// TwinCAT 3 PLC project _01_Observer
// ProgramVersion: 3.1.4023.0
// libraries:
//   Tc2_Standard, * (Beckhoff Automation GmbH)
//   Tc2_System, * (Beckhoff Automation GmbH)
//   Tc3_Module, * (Beckhoff Automation GmbH)
// project tree:
//   / MAIN.TcPOU, PlcTask.TcTTO
//   Observer Pattern/Pattern Base/ I_Observable.TcIO, I_Observer.TcIO, Observable.TcPOU
//   Observer Pattern/ P_ObserverPattern.TcPOU
//   Observer Pattern/Samples/ EventPublisherWithInheritance.TcPOU, EventPublisherWithComposition.TcPOU, FB_EventSubscriber.TcPOU, FB_EventSubscriber2.TcPOU, I_EventPublisher.TcIO
// (motion and I/O tree: see PLC project 13_decorator)
// real-time tasks:
//   TASK PlcTask: cycle T#10ms, priority 20, ADS port 350
// variable links:

CONFIGURATION _01_Observer
    RESOURCE PLC ON TwinCAT3
        TASK PlcTask(INTERVAL := T#10ms, PRIORITY := 20);
        PROGRAM MAIN WITH PlcTask : MAIN;
    END_RESOURCE
END_CONFIGURATION

// ---- Observer Pattern/Pattern Base/I_Observable.TcIO
INTERFACE I_Observable

METHOD Attach : bool
VAR_INPUT
	observer			: I_Observer;
END_VAR
END_METHOD

METHOD Detach : BOOL
VAR_INPUT
	observer			: I_Observer;
END_VAR
END_METHOD

END_INTERFACE

// ---- Observer Pattern/Pattern Base/I_Observer.TcIO
INTERFACE I_Observer

METHOD Update : BOOL
VAR_INPUT
END_VAR
END_METHOD

END_INTERFACE

// ---- Observer Pattern/Samples/I_EventPublisher.TcIO
INTERFACE I_EventPublisher EXTENDS I_Observable

PROPERTY Event : int
GET
END_GET
END_PROPERTY

END_INTERFACE

// ---- MAIN.TcPOU
PROGRAM MAIN
VAR
END_VAR

(* 
	GOF 		Define a one-to-many dependency between objects so that when one object changes state, 
				all its dependents are notified and updated automatically   
*)
P_ObserverPattern();

END_PROGRAM

// ---- Observer Pattern/P_ObserverPattern.TcPOU
PROGRAM P_ObserverPattern
VAR
	eventPublisher					: EventPublisherWithInheritance;
	eventPublisher2					: EventPublisherWithComposition;	
	
	eventSubscriber					: FB_EventSubscriber(eventPublisher);	
	eventSubscriber2				: FB_EventSubscriber2(eventPublisher2);	
	
	triggerEvent					: BOOL;
END_VAR

// Property changeEvent was only to be able to change the event from outside for the unit test
// Change according the use case of the observer
IF triggerEvent	THEN
	eventPublisher.changeEvent := eventPublisher.event + 1;
	eventPublisher2.changeEvent := eventPublisher2.event + 1;
	triggerEvent := FALSE;
END_IF
eventPublisher.CyclicCall();
eventPublisher2.CyclicCall();
eventSubscriber.CyclicCall();
eventSubscriber2.CyclicCall();

END_PROGRAM

// ---- Observer Pattern/Samples/EventPublisherWithInheritance.TcPOU
{attribute 'no_explicit_call' := 'FB_EventPublisher is a CLASS and must be accessed using methods or properties'}
FUNCTION_BLOCK EventPublisherWithInheritance EXTENDS Observable IMPLEMENTS I_EventPublisher
VAR
	_event							: INT;
	eventPrev						: INT;
END_VAR


// The body of a class must not be used for code.  
// Cyclic code should be called from a method if needed.

PROPERTY PUBLIC ChangeEvent : int
SET
// IMPLEMENTED ONLY FOR TESTING PURPOSES
VAR
END_VAR
_event := changeEvent;
END_SET
END_PROPERTY

METHOD CyclicCall
IF eventPrev <> _event 			THEN
	notify();
	eventPrev := _event;
END_IF
END_METHOD

// IMPLEMENTED ONLY FOR TESTING PURPOSES
PROPERTY Event : int
GET
event := _event;
END_GET
END_PROPERTY

END_FUNCTION_BLOCK

// ---- Observer Pattern/Pattern Base/Observable.TcPOU
{attribute 'no_explicit_call' := 'Observable is a CLASS and must be accessed using methods or properties'}
FUNCTION_BLOCK Observable IMPLEMENTS I_Observable
VAR
	verbose							: BOOL := TRUE;
	observers						: ARRAY[1..MAXOBSERVERS] OF I_Observer;
END_VAR
VAR CONSTANT
	MAXOBSERVERS					: INT := 5;		
END_VAR


// The body of a class must not be used for code.  
// Cyclic code should be called from a method if needed.

METHOD attach : BOOL
VAR_INPUT
	observer			: I_Observer;
END_VAR
VAR
	i					: INT;
END_VAR
(* default *)
attach := FALSE;

(* loop if the subscriber is already registered *)
FOR i := 1 TO MAXOBSERVERS DO
	IF observers[i] = observer 	THEN
		observer.update();
		attach := TRUE;
		RETURN;
	END_IF
END_FOR

(* loop for first free position if not yet attached *)
FOR i := 1 TO MAXOBSERVERS DO
	IF observers[i] = 0 	THEN
		observers[i] := observer;
		message('Observer registered');
		observer.update();
		attach := TRUE;
		EXIT;
	END_IF
END_FOR
END_METHOD

METHOD detach : BOOL
VAR_INPUT
	observer			: I_Observer;
END_VAR
VAR
	i					: INT;
END_VAR
(* default *)
detach := FALSE;

(* loop if the subscriber is already registered *)
FOR i := 1 TO MAXOBSERVERS DO
	IF observers[i] = observer 	THEN
		observers[i] := 0;
		message('Observer deregistered');
		detach := TRUE;
		RETURN;
	END_IF
END_FOR
END_METHOD

METHOD PRIVATE message : BOOL
VAR_INPUT
	strArg						: STRING;
END_VAR
// Log message
IF verbose  THEN
	ADSLOGSTR(
		msgCtrlMask := ADSLOG_MSGTYPE_HINT OR ADSLOG_MSGTYPE_LOG, // ADSLOG_MSGTYPE_ERROR OR ADSLOG_MSGTYPE_LOG, 
		msgFmtStr 	:= '%s',
		strArg 		:= strArg
		);
END_IF
END_METHOD

PROPERTY noOfAttachedObservers : int
GET
VAR
	i							: INT;
END_VAR
// In stead of using an internal counter that could fail
// run through the array of attached observers
(* loop for first free position if not yet attached *)
NoOfAttachedObservers := 0;
FOR i := 1 TO MAXOBSERVERS DO
	IF observers[i] <> 0 	THEN
		NoOfAttachedObservers := NoOfAttachedObservers + 1;
	END_IF
END_FOR
END_GET
END_PROPERTY

METHOD notify : BOOL
VAR
	i			: INT;
END_VAR
(* default *)
notify := FALSE;

(* loop if the subscriber is already registered *)
FOR i := 1 TO MAXOBSERVERS DO
	IF observers[i] <> 0 	THEN
		observers[i].update();
	END_IF
END_FOR
END_METHOD

END_FUNCTION_BLOCK

// ---- Observer Pattern/Samples/EventPublisherWithComposition.TcPOU
{attribute 'no_explicit_call' := 'FB_EventPublisher is a CLASS and must be accessed using methods or properties'}
FUNCTION_BLOCK EventPublisherWithComposition IMPLEMENTS I_EventPublisher
VAR
	_event							: INT;
	eventPrev						: INT;
	
	observable						: Observable;
END_VAR


// The body of a class must not be used for code.  
// Cyclic code should be called from a method if needed.

METHOD Attach : BOOL
VAR_INPUT
	observer	: I_Observer;
END_VAR
Attach := observable.Attach(observer);
END_METHOD

PROPERTY PUBLIC ChangeEvent : int
SET
// IMPLEMENTED ONLY FOR TESTING PURPOSES
VAR
END_VAR
_event := changeEvent;
END_SET
END_PROPERTY

METHOD CyclicCall
IF eventPrev <> _event 			THEN
	observable.Notify();
	eventPrev := _event;
END_IF
END_METHOD

METHOD Detach : BOOL
VAR_INPUT
	observer	: I_Observer;
END_VAR
Detach := observable.Detach(observer);
END_METHOD

// IMPLEMENTED ONLY FOR TESTING PURPOSES
PROPERTY Event : int
GET
event := _event;
END_GET
END_PROPERTY

END_FUNCTION_BLOCK

// ---- Observer Pattern/Samples/FB_EventSubscriber.TcPOU
{attribute 'no_explicit_call' := 'FB_EventSubscriber is a CLASS and must be accessed using methods or properties'}
FUNCTION_BLOCK FB_EventSubscriber IMPLEMENTS I_Observer
VAR	
	_eventPublisher					: I_EventPublisher;
	_event							: INT;
	
	verbose							: BOOL := TRUE;

	// Register after online change 
	registeredAtPublisher			: BOOL;	
END_VAR


// The body of a class must not be used for code.  
// Cyclic code should be called from a method if needed.

METHOD ChangePublisher
VAR_INPUT
	eventPublisher					: I_EventPublisher;
END_VAR
_eventPublisher := eventPublisher;
END_METHOD

METHOD cyclicCall
// Did we already register in the publisher?
IF NOT registeredAtPublisher	THEN
	registeredAtPublisher := _eventPublisher.attach(THIS^);
END_IF
END_METHOD

// IMPLEMENTED ONLY FOR TESTING PURPOSES
PROPERTY Event : int
GET
event := _event;
END_GET
END_PROPERTY

METHOD FB_init : BOOL
VAR_INPUT
	bInitRetains	 				: BOOL; // if TRUE, the retain variables are initialized (warm start / cold start)
	bInCopyCode 					: BOOL;  // if TRUE, the instance afterwards gets moved into the copy code (online change)
	EventPublisher					: I_EventPublisher;
END_VAR
_eventPublisher := eventPublisher;
END_METHOD

METHOD PRIVATE message : BOOL
VAR_INPUT
	dintArg						: DINT;
END_VAR
// Log message
IF verbose  THEN
	ADSLOGDINT(
		msgCtrlMask := ADSLOG_MSGTYPE_HINT OR ADSLOG_MSGTYPE_LOG, // ADSLOG_MSGTYPE_ERROR OR ADSLOG_MSGTYPE_LOG, 
		msgFmtStr 	:= 'Subscriber 1 knows the value changed to %d',
		dintArg 	:= dintArg
		);
END_IF
END_METHOD

METHOD Update : BOOL
// the publisher mentions an update, fetch the data
_event := _eventPublisher.event;
message(TO_DINT(_event));
END_METHOD

END_FUNCTION_BLOCK

// ---- Observer Pattern/Samples/FB_EventSubscriber2.TcPOU
{attribute 'no_explicit_call' := 'FB_EventSubscriber2 is a CLASS and must be accessed using methods or properties'}
FUNCTION_BLOCK FB_EventSubscriber2 IMPLEMENTS I_Observer
VAR	
	_eventPublisher					: I_EventPublisher;
	_event							: INT;
	
	verbose							: BOOL := TRUE;

	// Register after online change 
	registeredAtPublisher			: BOOL;
END_VAR

METHOD ChangePublisher
VAR_INPUT
	eventPublisher					: I_EventPublisher;
END_VAR
_eventPublisher := eventPublisher;
END_METHOD

METHOD CyclicCall
// Did we already register in the publisher?
IF NOT registeredAtPublisher	THEN
	registeredAtPublisher := _eventPublisher.attach(THIS^);
END_IF
END_METHOD

// IMPLEMENTED ONLY FOR TESTING PURPOSES
PROPERTY Event : int
GET
event := _event;
END_GET
END_PROPERTY

METHOD FB_init : BOOL
VAR_INPUT
	bInitRetains	 				: BOOL; // if TRUE, the retain variables are initialized (warm start / cold start)
	bInCopyCode 					: BOOL;  // if TRUE, the instance afterwards gets moved into the copy code (online change)
	eventPublisher					: I_EventPublisher;
END_VAR
_eventPublisher := eventPublisher;
END_METHOD

{attribute 'call_after_online_change_slot' := '0'}
METHOD PRIVATE fbreinit

(*	!!!!!!!!!!!!!!!!!!!!!!!!!!!!!!!!!
   	THIS METHOD is force called after every online change 
   	!= the fb_reinit system call that will be called after the instance of the concerned function block has been copied 
 	(during an online change after modifications in the function block declaration)

	This is necessary since both observer en observee have references to one other
	!!!!!!!!!!!!!!!!!!!!!!!!!!!!!!!!!	*)
registeredAtPublisher := FALSE;
breinit:=not breinit; // flip the test marker
END_METHOD

METHOD PRIVATE message : BOOL
VAR_INPUT
	dintArg						: DINT;
END_VAR
// Log message
IF verbose  THEN
	ADSLOGDINT(
		msgCtrlMask := ADSLOG_MSGTYPE_HINT OR ADSLOG_MSGTYPE_LOG, // ADSLOG_MSGTYPE_ERROR OR ADSLOG_MSGTYPE_LOG, 
		msgFmtStr 	:= 'Subscriber 2 knows the value changed to %d',
		dintArg 	:= dintArg
		);
END_IF
END_METHOD

METHOD Update : BOOL
// the publisher mentions an update, fetch the data
_event := _eventPublisher.event;
message(TO_DINT(_event));
END_METHOD

END_FUNCTION_BLOCK
